FUNCTION_BLOCK TestSocketAndPlug_Socket (* Template for a simple Basic Function Block Type *)
  (* Standard: 61499-2; Description: Copyright (c) 2019 Jan Holzweber This program and the accompanying materials are made available under the terms of the Eclipse Public License 2.0 which is available at https://www.eclipse.org/legal/epl-2.0/ SPDX-License-Identifier: EPL-2.0 *)
  (* Version 1.0, 2019-07-25, Jan Holzweber *)
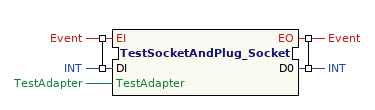
  EVENT_INPUT
    EI WITH DI; (* Normal Execution Request *)
  END_EVENT
  EVENT_OUTPUT
    EO WITH D0;
  END_EVENT
  VAR_INPUT
    DI : INT; (* Input event qualifier *)
  END_VAR
  VAR_OUTPUT
    D0 : INT;
  END_VAR
  SOCKETS
    TestAdapter : TestAdapter;
  END_SOCKETS
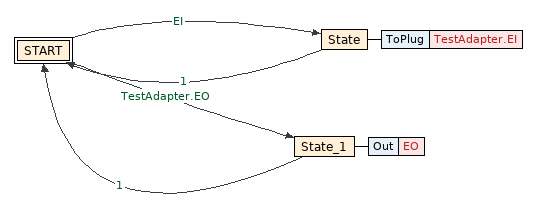
  EC_STATES
    START; (* Initial State *)
    State : ToPlug -> TestAdapter.EI;
    State_1 : Out -> EO;
  END_STATES
  EC_TRANSITIONS
    START TO State := EI;
    State TO START := 1;
    START TO State_1 := TestAdapter.EO;
    State_1 TO START := 1;
  END_TRANSITIONS
  ALGORITHM ToPlug IN ST: (* new algorithm *)
TestAdapter.DI := DI;
  END_ALGORITHM
  ALGORITHM Out IN ST: (* new algorithm *)
D0 := TestAdapter.D0;
  END_ALGORITHM
END_FUNCTION_BLOCK
